TYPE HMIHeader :
STRUCT
	PathOperatingMode	:	STRING;
	PathMachineState	:	STRING;
	NameApplication	:	STRING;
	ErrorIsActive	:	BOOL;
	State	:	INT;
END_STRUCT
END_TYPE

(* stored: Version 1.1.0.1
   DUT HMIHeader: Id {5cbe1d18-faa2-4d71-b308-6b6c7bfb6464} *)
